// TIA Portal V19 export
TYPE "typeVfdProduction"
// stored: Access Published
   STRUCT
      upperVel : Real;   // 产品模式速度上限
      lowVel : Real;   // 产品模式设定值，画面做限制根据上限值如果超了不允许输入
      highVel : Real;
   END_STRUCT;
END_TYPE
